(* CoDeSys 2.3 export: ALL.EXP *)
(* Libraries: ANALYZATION.LIB 5.10.99 08:05:06, G:\owen\dz_smarthome_lib.lib 9.5.15 16:30:44, G:\owen\lib\oscat_basic_333.lib 19.12.17 20:17:33, IECSFC.LIB 13.4.06 14:51:28, STANDARD.LIB 4.10.05 10:14:46, SysLibSockets.lib 20.2.06 13:31:14, SysLibTime.lib 20.2.06 13:31:16, Util.lib 18.5.10 14:14:28 *)

(* PLC configuration (modules and I/O channels)
PLC110_30 [Root] node -1, in %IB0 out %QB0 {param 1 = 1; param 2 = 1000; param 3 = 6}
  Fast discrete inputs [I_SIMPLE_INPUT] node 0, in %IB0 out %QB0 {param 1 = 10; param 9 = No}
    AT %IX0.0 [BitInput] Discrete input 1
    AT %IX0.1 [BitInput] Discrete input 2
  Discrete inputs - 16 [ID130] node 1, in %IB1 out %QB1 {param 1 = 1; param 9 = No; param 10 = 16}
    AT %IB1.0 [ByteInput] 8 discrete inputs
    AT %IB1.1 [ByteInput] 8 discrete inputs
  Fast discrete outputs [OWEN_ID570] node 2, in %IB2 out %QB2 {param 1 = FALSE; param 2 = FALSE; param 3 = FALSE; param 4 = FALSE; param 10 = No}
    RADIATOR_GUEST_OUT AT %QX2.0 [BitOutput] Fast discrete output 1 - radiator, guest room, 1 = OFF!
    RADIATOR_CHILDREN_NEAR_OUT AT %QX2.1 [BitOutput] Fast discrete output 2, radiator, children room, near the door, 1 = OFF
    RADIATOR_BEDROOM_OUT AT %QX2.2 [BitOutput] Fast discrete output 3
    RADIATOR_DINNER_OUT AT %QX2.3 [BitOutput] Fast discrete output 4 - dinner room radiator PWM, 0 = ON, 1 = OFF
  Discrete outputs - 8 [ID131] node 3, in %IB3 out %QB3 {param 1 = 0; param 4 = No; param 5 = 10}
    AT %QB3.0 [ByteOutput] 8 discrete outputs
  Special input [ID103] node 4, in %IB4 out %QB4 {param 1 = 1000; param 2 = 1; param 3 = 400; param 4 = 3000; param 5 = No}
    AT %IX4.0 [BitInput] Special input
  Special output [ID104] node 5, in %IB5 out %QB5 {param 1 = No; param 2 = 1}
    AT %QX5.0 [BitOutput] Special output
  ModBus (Master) [MODBUS_MASTER_ID450] node 6, in %IB6 out %QB6 {param 1 = No}
    AT %QD6.0 [DWordOutput] Last address
    AT %QW6.1 [WordOutput] Last error
    RS-485-1 [COM1_USART] node 0, in %IB6.0 out %QB6.0 {param 1 = 11520; param 2 = NO PARITY CHECK; param 3 = 8 bits; param 4 = One stop bit; param 5 = RS485; param 6 = ASCII; param 7 = 0; param 8 = No}
    OWEN_MVA8 [ID2050] node 1, in %IB6.1 out %QB6.1 {param 1 = 10:0:0:223; param 2 = 30; param 3 = 502; param 4 = Serial; param 5 = 80; param 6 = By poll time; param 7 = 400; param 8 = No; param 9 = 0; param 10 = Trace_mode}
      mva8_0_cmd AT %QB6.1.0 [ComChannel] Command (0xff - Start)
      Cycle time measuring on input 1 [ID2066] node 0, in %IB6.1.0 out %QB6.1.0 {param 1 = 3; param 2 = Command Read (03); param 7 = No}
        AT %IW6.1.0.0 [WordInput]
      Value in input 1 [ID2067] node 1, in %IB6.1.1 out %QB6.1.1 {param 1 = 4; param 2 = Command Read (03); param 7 = No}
        mva0_t0 AT %ID6.1.1.0 [FloatInput]
      Cycle time measuring on input 2 [ID2068] node 2, in %IB6.1.2 out %QB6.1.2 {param 1 = 9; param 2 = Command Read (03); param 7 = No}
        AT %IW6.1.2.0 [WordInput]
      Value in input 2 [ID2069] node 3, in %IB6.1.3 out %QB6.1.3 {param 1 = 10; param 2 = Command Read (03); param 7 = No}
        mva0_t1 AT %ID6.1.3.0 [FloatInput]
      Cycle time measuring on input 3 [ID2070] node 4, in %IB6.1.4 out %QB6.1.4 {param 1 = 15; param 2 = Command Read (03); param 7 = No}
        AT %IW6.1.4.0 [WordInput]
      Value in input 3 [ID2071] node 5, in %IB6.1.5 out %QB6.1.5 {param 1 = 16; param 2 = Command Read (03); param 7 = No}
        mva0_t2 AT %ID6.1.5.0 [FloatInput]
      Cycle time measuring on input 4 [ID2072] node 6, in %IB6.1.6 out %QB6.1.6 {param 1 = 21; param 2 = Command Read (03); param 7 = No}
        AT %IW6.1.6.0 [WordInput]
      Value in input 4 [ID2073] node 7, in %IB6.1.7 out %QB6.1.7 {param 1 = 22; param 2 = Command Read (03); param 7 = No}
        mva0_t3 AT %ID6.1.7.0 [FloatInput]
      Cycle time measuring on input 5 [ID2074] node 8, in %IB6.1.8 out %QB6.1.8 {param 1 = 27; param 2 = Command Read (03); param 7 = No}
        AT %IW6.1.8.0 [WordInput]
      Value in input 5 [ID2075] node 9, in %IB6.1.9 out %QB6.1.9 {param 1 = 28; param 2 = Command Read (03); param 7 = No}
        mva0_t4 AT %ID6.1.9.0 [FloatInput]
      Cycle time measuring on input 6 [ID2076] node 10, in %IB6.1.10 out %QB6.1.10 {param 1 = 33; param 2 = Command Read (03); param 7 = No}
        AT %IW6.1.10.0 [WordInput]
      Value in input 6 [ID2077] node 11, in %IB6.1.11 out %QB6.1.11 {param 1 = 34; param 2 = Command Read (03); param 7 = No}
        mva0_t5 AT %ID6.1.11.0 [FloatInput]
      Cycle time measuring on input 7 [ID2078] node 12, in %IB6.1.12 out %QB6.1.12 {param 1 = 39; param 2 = Command Read (03); param 7 = No}
        AT %IW6.1.12.0 [WordInput]
      Value in input 7 [ID2079] node 13, in %IB6.1.13 out %QB6.1.13 {param 1 = 40; param 2 = Command Read (03); param 7 = No}
        mva0_t6 AT %ID6.1.13.0 [FloatInput]
      Cycle time measuring on input 8 [ID2080] node 14, in %IB6.1.14 out %QB6.1.14 {param 1 = 45; param 2 = Command Read (03); param 7 = No}
        AT %IW6.1.14.0 [WordInput]
      Value in input 8 [ID2081] node 15, in %IB6.1.15 out %QB6.1.15 {param 1 = 46; param 2 = Command Read (03); param 7 = No}
        mva0_t7 AT %ID6.1.15.0 [FloatInput]
    OWEN_MVA8 [ID2050] node 2, in %IB6.2 out %QB6.2 {param 1 = 10:0:0:223; param 2 = 30; param 3 = 502; param 4 = Serial; param 5 = 88; param 6 = By poll time; param 7 = 400; param 8 = No; param 9 = 0; param 10 = Trace_mode}
      mva8_1_cmd AT %QB6.2.0 [ComChannel] Command (0xff - Start)
      Cycle time measuring on input 1 [ID2066] node 0, in %IB6.2.0 out %QB6.2.0 {param 1 = 3; param 2 = Command Read (03); param 7 = No}
        AT %IW6.2.0.0 [WordInput]
      Value in input 1 [ID2067] node 1, in %IB6.2.1 out %QB6.2.1 {param 1 = 4; param 2 = Command Read (03); param 7 = No}
        mva1_t0 AT %ID6.2.1.0 [FloatInput]
      Cycle time measuring on input 2 [ID2068] node 2, in %IB6.2.2 out %QB6.2.2 {param 1 = 9; param 2 = Command Read (03); param 7 = No}
        AT %IW6.2.2.0 [WordInput]
      Value in input 2 [ID2069] node 3, in %IB6.2.3 out %QB6.2.3 {param 1 = 10; param 2 = Command Read (03); param 7 = No}
        mva1_t1 AT %ID6.2.3.0 [FloatInput]
      Cycle time measuring on input 3 [ID2070] node 4, in %IB6.2.4 out %QB6.2.4 {param 1 = 15; param 2 = Command Read (03); param 7 = No}
        AT %IW6.2.4.0 [WordInput]
      Value in input 3 [ID2071] node 5, in %IB6.2.5 out %QB6.2.5 {param 1 = 16; param 2 = Command Read (03); param 7 = No}
        mva1_t2 AT %ID6.2.5.0 [FloatInput]
      Cycle time measuring on input 4 [ID2072] node 6, in %IB6.2.6 out %QB6.2.6 {param 1 = 21; param 2 = Command Read (03); param 7 = No}
        AT %IW6.2.6.0 [WordInput]
      Value in input 4 [ID2073] node 7, in %IB6.2.7 out %QB6.2.7 {param 1 = 22; param 2 = Command Read (03); param 7 = No}
        mva1_t3 AT %ID6.2.7.0 [FloatInput]
      Cycle time measuring on input 5 [ID2074] node 8, in %IB6.2.8 out %QB6.2.8 {param 1 = 27; param 2 = Command Read (03); param 7 = No}
        AT %IW6.2.8.0 [WordInput]
      Value in input 5 [ID2075] node 9, in %IB6.2.9 out %QB6.2.9 {param 1 = 28; param 2 = Command Read (03); param 7 = No}
        mva1_t4 AT %ID6.2.9.0 [FloatInput]
      Cycle time measuring on input 6 [ID2076] node 10, in %IB6.2.10 out %QB6.2.10 {param 1 = 33; param 2 = Command Read (03); param 7 = No}
        AT %IW6.2.10.0 [WordInput]
      Value in input 6 [ID2077] node 11, in %IB6.2.11 out %QB6.2.11 {param 1 = 34; param 2 = Command Read (03); param 7 = No}
        mva1_t5 AT %ID6.2.11.0 [FloatInput]
      Cycle time measuring on input 7 [ID2078] node 12, in %IB6.2.12 out %QB6.2.12 {param 1 = 39; param 2 = Command Read (03); param 7 = No}
        AT %IW6.2.12.0 [WordInput]
      Value in input 7 [ID2079] node 13, in %IB6.2.13 out %QB6.2.13 {param 1 = 40; param 2 = Command Read (03); param 7 = No}
        mva1_t6 AT %ID6.2.13.0 [FloatInput]
      Cycle time measuring on input 8 [ID2080] node 14, in %IB6.2.14 out %QB6.2.14 {param 1 = 45; param 2 = Command Read (03); param 7 = No}
        AT %IW6.2.14.0 [WordInput]
      Value in input 8 [ID2081] node 15, in %IB6.2.15 out %QB6.2.15 {param 1 = 46; param 2 = Command Read (03); param 7 = No}
        mva1_t7 AT %ID6.2.15.0 [FloatInput]
    OWEN_MVA8 [ID2050] node 3, in %IB6.3 out %QB6.3 {param 1 = 10:0:0:223; param 2 = 30; param 3 = 502; param 4 = Serial; param 5 = 96; param 6 = By poll time; param 7 = 400; param 8 = No; param 9 = 0; param 10 = Trace_mode}
      mva8_2_cmd AT %QB6.3.0 [ComChannel] Command (0xff - Start)
      Cycle time measuring on input 1 [ID2066] node 0, in %IB6.3.0 out %QB6.3.0 {param 1 = 3; param 2 = Command Read (03); param 7 = No}
        AT %IW6.3.0.0 [WordInput]
      Value in input 1 [ID2067] node 1, in %IB6.3.1 out %QB6.3.1 {param 1 = 4; param 2 = Command Read (03); param 7 = No}
        mva2_t0 AT %ID6.3.1.0 [FloatInput]
      Cycle time measuring on input 2 [ID2068] node 2, in %IB6.3.2 out %QB6.3.2 {param 1 = 9; param 2 = Command Read (03); param 7 = No}
        AT %IW6.3.2.0 [WordInput]
      Value in input 2 [ID2069] node 3, in %IB6.3.3 out %QB6.3.3 {param 1 = 10; param 2 = Command Read (03); param 7 = No}
        mva2_t1 AT %ID6.3.3.0 [FloatInput]
      Cycle time measuring on input 3 [ID2070] node 4, in %IB6.3.4 out %QB6.3.4 {param 1 = 15; param 2 = Command Read (03); param 7 = No}
        AT %IW6.3.4.0 [WordInput]
      Value in input 3 [ID2071] node 5, in %IB6.3.5 out %QB6.3.5 {param 1 = 16; param 2 = Command Read (03); param 7 = No}
        mva2_t2 AT %ID6.3.5.0 [FloatInput]
      Cycle time measuring on input 4 [ID2072] node 6, in %IB6.3.6 out %QB6.3.6 {param 1 = 21; param 2 = Command Read (03); param 7 = No}
        AT %IW6.3.6.0 [WordInput]
      Value in input 4 [ID2073] node 7, in %IB6.3.7 out %QB6.3.7 {param 1 = 22; param 2 = Command Read (03); param 7 = No}
        mva2_t3 AT %ID6.3.7.0 [FloatInput]
      Cycle time measuring on input 5 [ID2074] node 8, in %IB6.3.8 out %QB6.3.8 {param 1 = 27; param 2 = Command Read (03); param 7 = No}
        AT %IW6.3.8.0 [WordInput]
      Value in input 5 [ID2075] node 9, in %IB6.3.9 out %QB6.3.9 {param 1 = 28; param 2 = Command Read (03); param 7 = No}
        mva2_t4 AT %ID6.3.9.0 [FloatInput]
      Cycle time measuring on input 6 [ID2076] node 10, in %IB6.3.10 out %QB6.3.10 {param 1 = 33; param 2 = Command Read (03); param 7 = No}
        AT %IW6.3.10.0 [WordInput]
      Value in input 6 [ID2077] node 11, in %IB6.3.11 out %QB6.3.11 {param 1 = 34; param 2 = Command Read (03); param 7 = No}
        mva2_t5 AT %ID6.3.11.0 [FloatInput]
      Cycle time measuring on input 7 [ID2078] node 12, in %IB6.3.12 out %QB6.3.12 {param 1 = 39; param 2 = Command Read (03); param 7 = No}
        AT %IW6.3.12.0 [WordInput]
      Value in input 7 [ID2079] node 13, in %IB6.3.13 out %QB6.3.13 {param 1 = 40; param 2 = Command Read (03); param 7 = No}
        mva2_t6 AT %ID6.3.13.0 [FloatInput]
      Cycle time measuring on input 8 [ID2080] node 14, in %IB6.3.14 out %QB6.3.14 {param 1 = 45; param 2 = Command Read (03); param 7 = No}
        AT %IW6.3.14.0 [WordInput]
      Value in input 8 [ID2081] node 15, in %IB6.3.15 out %QB6.3.15 {param 1 = 46; param 2 = Command Read (03); param 7 = No}
        mva2_t7 AT %ID6.3.15.0 [FloatInput]
  ModBus (Master) [MODBUS_MASTER_ID450] node 7, in %IB7 out %QB7 {param 1 = No}
    AT %QD7.0 [DWordOutput] Last address
    AT %QW7.1 [WordOutput] Last error
    RS-485-2 [COM3_USART] node 0, in %IB7.0 out %QB7.0 {param 1 = 9600; param 2 = NO PARITY CHECK; param 3 = 8 bits; param 4 = One stop bit; param 5 = RS485; param 6 = RTU; param 7 = 0; param 8 = No}
    Universal Modbus device [ID2000] node 1, in %IB7.1 out %QB7.1 {param 1 = 10:0:0:223; param 2 = 150; param 3 = 502; param 4 = Serial; param 5 = 16; param 6 = By value change; param 7 = 200; param 8 = No; param 9 = 0; param 10 = Trace_mode}
      z033_special_cmd AT %QB7.1.0 [ComChannel] Command (0xff - Start)
      Register output module [ID2004] node 0, in %IB7.1.0 out %QB7.1.0 {param 1 = 16#116; param 2 = Preset singl register (0x06); param 8 = No}
        z033_hum116_out AT %QW7.1.0.0 [WordOutput]
      Register output module [ID2004] node 1, in %IB7.1.1 out %QB7.1.1 {param 1 = 16#115; param 2 = Preset singl register (0x06); param 8 = No}
        z033_temperature115_out AT %QW7.1.1.0 [WordOutput]
    Universal Modbus device [ID2000] node 2, in %IB7.2 out %QB7.2 {param 1 = 10:0:0:223; param 2 = 150; param 3 = 502; param 4 = Serial; param 5 = 16; param 6 = Both; param 7 = 200; param 8 = No; param 9 = 0; param 10 = Trace_mode}
      z033_cmd AT %QB7.2.0 [ComChannel] Command (0xff - Start)
      Register output module [ID2004] node 0, in %IB7.2.0 out %QB7.2.0 {param 1 = 16#112; param 2 = Preset singl register (0x06); param 8 = No}
        z033_Setup112 AT %QW7.2.0.0 [WordOutput]
      Register output module [ID2004] node 1, in %IB7.2.1 out %QB7.2.1 {param 1 = 16#113; param 2 = Preset singl register (0x06); param 8 = No}
        z033_Setup113 AT %QW7.2.1.0 [WordOutput]
      Register input module [ID2003] node 2, in %IB7.2.2 out %QB7.2.2 {param 1 = 16#114; param 2 = Read holding Registers  (0x03); param 8 = No}
        z033_mode114_in AT %IW7.2.2.0 [WordInput]
      Register output module [ID2004] node 3, in %IB7.2.3 out %QB7.2.3 {param 1 = 16#114; param 2 = Preset singl register (0x06); param 8 = No}
        z033_mode114_out AT %QW7.2.3.0 [WordOutput]
      Register input module [ID2003] node 4, in %IB7.2.4 out %QB7.2.4 {param 1 = 16#115; param 2 = Read holding Registers  (0x03); param 8 = No}
        z033_temperature115_in AT %IW7.2.4.0 [WordInput]
      Register input module [ID2003] node 5, in %IB7.2.5 out %QB7.2.5 {param 1 = 16#116; param 2 = Read holding Registers  (0x03); param 8 = No}
        z033_hum116_in AT %IW7.2.5.0 [WordInput]
      Register input module [ID2003] node 6, in %IB7.2.6 out %QB7.2.6 {param 1 = 16#117; param 2 = Read holding Registers  (0x03); param 8 = No}
        z033_room_temp117_in AT %IW7.2.6.0 [WordInput] temp measured by panel, no set
      Register output module [ID2004] node 7, in %IB7.2.7 out %QB7.2.7 {param 1 = 16#118; param 2 = Preset singl register (0x06); param 8 = No}
        z033_floor_temp118_out AT %QW7.2.7.0 [WordOutput]
      Register output module [ID2004] node 8, in %IB7.2.8 out %QB7.2.8 {param 1 = 16#119; param 2 = Preset singl register (0x06); param 8 = No}
        z033_outdoor_hum119_out AT %QW7.2.8.0 [WordOutput]
      Register output module [ID2004] node 9, in %IB7.2.9 out %QB7.2.9 {param 1 = 16#11A; param 2 = Preset singl register (0x06); param 8 = No}
        z033_room_hum11a_out AT %QW7.2.9.0 [WordOutput]
      Register output module [ID2004] node 10, in %IB7.2.10 out %QB7.2.10 {param 1 = 16#11B; param 2 = Preset singl register (0x06); param 8 = No}
        z033_air_hum11b_out AT %QW7.2.10.0 [WordOutput]
      Register output module [ID2004] node 11, in %IB7.2.11 out %QB7.2.11 {param 1 = 16#11c; param 2 = Preset singl register (0x06); param 8 = No}
        z033_errmode11c_out AT %QW7.2.11.0 [WordOutput]
      Register output module [ID2004] node 12, in %IB7.2.12 out %QB7.2.12 {param 1 = 16#11D; param 2 = Preset singl register (0x06); param 8 = No}
        z033_clock11d_out AT %QW7.2.12.0 [WordOutput]
      Register input module [ID2003] node 13, in %IB7.2.13 out %QB7.2.13 {param 1 = 16#11C; param 2 = Read holding Registers  (0x03); param 8 = No}
        z033_errmode11c_in AT %IW7.2.13.0 [WordInput]
      Register output module [ID2004] node 14, in %IB7.2.14 out %QB7.2.14 {param 1 = 16#117; param 2 = Preset singl register (0x06); param 8 = No}
        z033_air_temp_117_out AT %QW7.2.14.0 [WordOutput]
  Button [ID003] node 8, in %IB8 out %QB8
    AT %IX8.0 [BitInput] Button Start/Stop
  ModBus (slave) [MODBUS_ID400] node 9, in %IB9 out %QB9 {param 1 = 1; param 2 = No}
    Modbus [MODBUS_ID302] node 0, in %IB9.0 out %QB9.0
      TCP [TCP_ID221] node 0, in %IB9.0.0 out %QB9.0.0 {param 1 = 502; param 2 = No}
    2 byte [Register] node 1, in %IB9.1 out %QB9.1
      Uplink_Target_Temp AT %QW9.1.0 [WordOutput]
    2 byte [Register] node 2, in %IB9.2 out %QB9.2
      Uplink_Target_Humid AT %QW9.2.0 [WordOutput]
  ModBus (Master) [MODBUS_MASTER_ID450] node 10, in %IB10 out %QB10 {param 1 = No}
    AT %QD10.0 [DWordOutput] Last address
    AT %QW10.1 [WordOutput] Last error
    Debug RS-232 [DEBUG_USART] node 0, in %IB10.0 out %QB10.0 {param 1 = 11520; param 2 = NO PARITY CHECK; param 3 = 8 bits; param 4 = One stop bit; param 5 = RS232; param 6 = ASCII; param 7 = 0; param 8 = No}
    Universal Modbus device [ID2000] node 1, in %IB10.1 out %QB10.1 {param 1 = 192:168:88:130; param 2 = 150; param 3 = 502; param 4 = TCP; param 5 = 1; param 6 = By poll time; param 7 = 2000; param 8 = No; param 9 = 0; param 10 = Trace_mode}
      dz1w_cmd AT %QB10.1.0 [ComChannel] Command (0xff - Start)
      Register input module [ID2003] node 0, in %IB10.1.0 out %QB10.1.0 {param 1 = 1024; param 2 = Read holding Registers  (0x03); param 8 = No}
        sensor_id0 AT %IW10.1.0.0 [WordInput]
      Register input module [ID2003] node 1, in %IB10.1.1 out %QB10.1.1 {param 1 = 1025; param 2 = Read holding Registers  (0x03); param 8 = No}
        sensor_id1 AT %IW10.1.1.0 [WordInput]
      Register input module [ID2003] node 2, in %IB10.1.2 out %QB10.1.2 {param 1 = 1026; param 2 = Read holding Registers  (0x03); param 8 = No}
        sensor_id2 AT %IW10.1.2.0 [WordInput]
      Register input module [ID2003] node 3, in %IB10.1.3 out %QB10.1.3 {param 1 = 1027; param 2 = Read holding Registers  (0x03); param 8 = No}
        sensor_id3 AT %IW10.1.3.0 [WordInput]
      Register input module [ID2003] node 4, in %IB10.1.4 out %QB10.1.4 {param 1 = 1028; param 2 = Read holding Registers  (0x03); param 8 = No}
        sensor_id4 AT %IW10.1.4.0 [WordInput]
      Register input module [ID2003] node 5, in %IB10.1.5 out %QB10.1.5 {param 1 = 1029; param 2 = Read holding Registers  (0x03); param 8 = No}
        sensor_id5 AT %IW10.1.5.0 [WordInput]
      Register input module [ID2003] node 6, in %IB10.1.6 out %QB10.1.6 {param 1 = 1030; param 2 = Read holding Registers  (0x03); param 8 = No}
        sensor_id6 AT %IW10.1.6.0 [WordInput]
      Register input module [ID2003] node 7, in %IB10.1.7 out %QB10.1.7 {param 1 = 1031; param 2 = Read holding Registers  (0x03); param 8 = No}
        sensor_id7 AT %IW10.1.7.0 [WordInput]
      Register input module [ID2003] node 8, in %IB10.1.8 out %QB10.1.8 {param 1 = 1032; param 2 = Read holding Registers  (0x03); param 8 = No}
        sensor_id8 AT %IW10.1.8.0 [WordInput]
      Register input module [ID2003] node 9, in %IB10.1.9 out %QB10.1.9 {param 1 = 1033; param 2 = Read holding Registers  (0x03); param 8 = No}
        sensor_id9 AT %IW10.1.9.0 [WordInput]
      Register input module [ID2003] node 10, in %IB10.1.10 out %QB10.1.10 {param 1 = 1034; param 2 = Read holding Registers  (0x03); param 8 = No}
        sensor_id10 AT %IW10.1.10.0 [WordInput]
      Register input module [ID2003] node 11, in %IB10.1.11 out %QB10.1.11 {param 1 = 2048; param 2 = Read holding Registers  (0x03); param 8 = No}
        seq_sensor_0 AT %IW10.1.11.0 [WordInput]
      Register input module [ID2003] node 12, in %IB10.1.12 out %QB10.1.12 {param 1 = 2049; param 2 = Read holding Registers  (0x03); param 8 = No}
        seq_sensor_1 AT %IW10.1.12.0 [WordInput]
*)

(* Task configuration *)
TASK OnceASecond (PRIORITY := 1, INTERVAL := T#1s0ms);
ONCE_A_SECOND_PRG();
END_TASK
TASK HTTP_POLLER (PRIORITY := 5, INTERVAL := T#1s0ms);
TCP_POLL();
END_TASK
TASK Main (PRIORITY := 2, INTERVAL := T#50ms);
PLC_PRG();
END_TASK
TASK MQTT (PRIORITY := 4, INTERVAL := T#1s0ms);
MQTT_MAIN();
END_TASK

(* Global variable list: Global_Variables *)
VAR_GLOBAL RETAIN PERSISTENT


	GLOBAL_Target_Room_Temp				: REAL := 26;
	GLOBAL_Target_Room_Humid				: REAL := 30;

	GLOBAL_Current_Entrance_Air_Temp		: REAL	:= 0;
	GLOBAL_Current_Entrance_Floor_Temp	: REAL := 100;

	GLOBAL_Current_Bath_Air_Temp			: REAL	:= 0;
	GLOBAL_Current_Bath_Floor_Temp		: REAL := 100;

	GLOBAL_Current_Bath_Tube_Temp		: REAL := 0;

	GLOBAL_Current_Dinner_Air_Temp			: REAL	:= 0;		(* Composite made of 3 sensors, used to control floor *)
	GLOBAL_Current_Dinner_Floor_Temp		: REAL := 100;

	GLOBAL_Current_Dinner_Air_Bottom_Temp			: REAL	:= 0; (* Bottom sensor, near the radiator *)
	GLOBAL_Current_Dinner_Air_Middle_Temp			: REAL	:= 0; (* Middle sensor, in the z033 panel, 1 degree step *)

	GLOBAL_Current_Guest_Air_Temp			: REAL := 0;

	GLOBAL_Current_Kitchen_Air_Ceiling_Temp			: REAL	:= 0; (* Ceiling sensor, in the fire sensor, kitchen *)

	GLOBAL_Current_Children_Air_Temp		: REAL	:= 0;
	GLOBAL_Current_Children_Floor_Temp	: REAL := 100;

	GLOBAL_Current_Badroom_Air_Temp		: REAL	:= 0;

	GLOBAL_Current_Bath_Air_Humid			: REAL := 0;

	GLOBAL_Current_Outdoor_Air_Temp		: REAL := 0;


END_VAR



VAR_GLOBAL CONSTANT
	SANE_TEMP_MIN: REAL := 10;		(*Minimum temp value assumed to be sane*)
	SANE_TEMP_MAX: REAL := 40;		(*Maximum temp value assumed to be sane*)

	SANE_HUMID_MIN:	WORD		:= 15;
	SANE_HUMID_MAX:	WORD		:= 55;

END_VAR

(* POU ONCE_A_SECOND_PRG, ST *)
PROGRAM ONCE_A_SECOND_PRG

VAR

	FLOOR_ENTRANCE		: FLOOR_PID;
	FLOOR_BATH				: FLOOR_PID;
	(*FLOOR_DINNER			: FLOOR_PID;*)
	DINNER_PID			: DUAL_PID;
	(*FLOOR_CHILDREN		: FLOOR_PID;*)
	CHILDREN_PID			: DUAL_PID;
	GUEST_PID			: DUAL_PID;

	PWM_ENTRANCE		: PWM;
	PWM_BATH				: PWM;
	PWM_DINNER			: PWM;
	PWM_CHILDREN			: PWM;

(*	PWM_DINNER_RADIATOR		: PWM; *)
	PWM_DINNER_RADIATOR		: RADIATOR_PWM;
	PWM_GUEST_RADIATOR		: RADIATOR_PWM;
	PWM_CHILDREN_RADIATOR	: RADIATOR_PWM;


END_VAR
	(* Must be called once a second! *)



	(* Entrance *)

	FLOOR_ENTRANCE( Target := GLOBAL_Target_Room_Temp, Current := GLOBAL_Current_Entrance_Air_Temp, Floor := GLOBAL_Current_Entrance_Floor_Temp );

	PWM_ENTRANCE( DUTY := FLOOR_ENTRANCE.DUTY, PHASE_SHIFT := 0 );

	HEAT_ENTRANCE_OUT := PWM_ENTRANCE.OUT_ON;



	(* Bath *)

	FLOOR_BATH( Target := GLOBAL_Target_Room_Temp, Current := GLOBAL_Current_Bath_Air_Temp, Floor := GLOBAL_Current_Bath_Floor_Temp );

	PWM_BATH( DUTY := FLOOR_BATH.DUTY, PHASE_SHIFT := 2 );

	HEAT_BATH_OUT := PWM_BATH.OUT_ON;


	(* Dinner *)

(*
	FLOOR_DINNER( Target := GLOBAL_Target_Room_Temp, Current := GLOBAL_Current_Dinner_Air_Temp, Floor := GLOBAL_Current_Dinner_Floor_Temp );
*)
	DINNER_PID( Target := GLOBAL_Target_Room_Temp, Current := GLOBAL_Current_Dinner_Air_Temp, Floor := GLOBAL_Current_Dinner_Floor_Temp );

	PWM_DINNER( DUTY := DINNER_PID.FLOOR_DUTY, PHASE_SHIFT := 4 );

	PWM_DINNER_RADIATOR( DUTY := DINNER_PID.RADIATOR_DUTY, PHASE_SHIFT := 0 );

	HEAT_DINNER_OUT := PWM_DINNER.OUT_ON;

	RADIATOR_DINNER_OUT := NOT PWM_DINNER_RADIATOR.OUT_ON; (* Naive impl - just control radiator just like floor *)

	(* Guest - no hot floor *)

	GUEST_PID( Target := GLOBAL_Target_Room_Temp, Current := GLOBAL_Current_Guest_Air_Temp, Floor := 50 ); (* no floor, give insane input value *)
	PWM_GUEST_RADIATOR( DUTY := GUEST_PID.RADIATOR_DUTY, PHASE_SHIFT := 0 );
	RADIATOR_GUEST_OUT := NOT PWM_GUEST_RADIATOR.OUT_ON; (* Naive impl - just control radiator just like floor *)

	(* Children *)

	(* FLOOR_CHILDREN( Target := GLOBAL_Target_Room_Temp, Current := GLOBAL_Current_CHILDREN_Air_Temp, Floor := GLOBAL_Current_CHILDREN_Floor_Temp ); *)

	CHILDREN_PID(        Target := GLOBAL_Target_Room_Temp, Current := GLOBAL_Current_CHILDREN_Air_Temp, Floor := GLOBAL_Current_CHILDREN_Floor_Temp );

	(*PWM_CHILDREN( DUTY := FLOOR_CHILDREN.DUTY, PHASE_SHIFT := 6 );*)
	PWM_CHILDREN( DUTY := CHILDREN_PID.FLOOR_DUTY, PHASE_SHIFT := 6 );


	PWM_CHILDREN_RADIATOR( DUTY := CHILDREN_PID.RADIATOR_DUTY, PHASE_SHIFT := 0 );

	HEAT_CHILDREN_OUT := PWM_CHILDREN.OUT_ON;

	RADIATOR_CHILDREN_NEAR_OUT := NOT PWM_CHILDREN_RADIATOR.OUT_ON;
END_PROGRAM

(* POU PID-PWM/FLOOR_PID, ST *)
FUNCTION_BLOCK FLOOR_PID

VAR_INPUT
	Target			: REAL;		(* Уставка, target ROOM temperature value to achieve *)
	Current		: REAL;		(* Current measured ROOM temperature value *)

	Floor			: REAL;		(* Current measured FLOOR temperature value *)
	Limited		: REAL := 35;	(* maximum FLOOR temperature value not to overcome*)


END_VAR

VAR_OUTPUT

	DUTY				: INT;		(* Duty cycle for heater *)

END_VAR

VAR

	TMP				: INT;
(*
	INTEGRAL			: INT;
*)
END_VAR
(*

	Actually we have TWO regulators here, one is PID (or PI) - for room temperature,
	and one is simple limiting for floor temperature.

*)

	(* room temp seems to be insane, use floor temp instead *)
	IF Current < 1 THEN
		Current := Floor;
	END_IF


	(* Simple FLOOR temp limit *)

	IF Floor > Limited THEN
		DUTY := 0;
		RETURN;
	END_IF

	(* TEMPORARY IMPL! *)

	IF Current > Target THEN
		DUTY := 0;
		RETURN;
	END_IF

	TMP := REAL_TO_INT(  (Target - Current) * 100 / 4 ); (* 4 degrees of difference mean 100% of power *)

	IF TMP < 0 THEN
		TMP := 0;
	END_IF

	IF TMP > 100 THEN
		TMP := 100;
	END_IF

	DUTY := TMP;
END_FUNCTION_BLOCK

(* POU PID-PWM/DUAL_PID, ST *)
FUNCTION_BLOCK DUAL_PID

VAR_INPUT
	Target			: REAL;		(* Уставка, target ROOM temperature value to achieve *)
	Current		: REAL;		(* Current measured ROOM temperature value *)

	Floor			: REAL;		(* Current measured FLOOR temperature value *)
	Limited		: REAL := 33;	(* Maximum FLOOR temperature value not to overcome*)


END_VAR

VAR_OUTPUT

	FLOOR_DUTY				: INT;		(* Duty cycle for floor heater *)
	RADIATOR_DUTY				: INT;		(* Duty cycle for wall radiator *)

END_VAR

VAR

	LINEAR			: INT;
	INTEGRAL			: REAL;		(* +- 1000 *)
	DIFFERENTIAL 	: REAL;		(* +- 100 *)
	DUTY				: INT;		(* Duty cycle - total *)

	Diff_Timer			: INT;
	Diff_Prev_Temp	: REAL		:= -1000;
	Diff_Temp_Delta	: REAL;		(* Difference of temperature in one minute *)
	Diff_Sane 			: BOOL;

END_VAR


VAR CONSTANT

	ONLY_RADIATOR_DUTY_LIMIT	: INT := 20;

	Diff_Timer_Time					: INT := 120;

END_VAR
(*

	Actually we have TWO regulators here, one is PID (or PI) - for room temperature,
	and one is simple limiting for floor temperature.

*)

	(* room temp seems to be insane, use floor temp instead *)
	IF Current < 1 THEN
		Current := Floor;
	END_IF




	LINEAR := REAL_TO_INT(  (Target - Current) * 100 / 4 ); (* 4 degrees of difference mean 100% of power *)
	LINEAR := REAL_TO_INT( LIMIT_VALUE( LINEAR, -100, 100) );

	(* Integral part *)

	INTEGRAL := INTEGRAL + (LINEAR / 2500.0); (* integration time about 0,65 hr *)

	INTEGRAL := LIMIT_VALUE( INTEGRAL, -100, 100 );

	(* Diff part *)

	Diff_Sane := TRUE;

	Diff_Timer := Diff_Timer + 1;
	IF Diff_Timer >= Diff_Timer_Time THEN
		Diff_Timer := 0;

		IF NOT IS_SANE_TEMP( Diff_Prev_Temp ) THEN
			Diff_Sane := FALSE;
		END_IF

		Diff_Temp_Delta := Current - Diff_Prev_Temp;
		Diff_Prev_Temp := Current;

	END_IF

	IF NOT Diff_Sane THEN
		Diff_Temp_Delta := 0;
	END_IF

	(* MINUS 0.5 degree per 2 minutes is 400% of power *)
	DIFFERENTIAL := - Diff_Temp_Delta * 200 * 4;

	(* Limit diff part to 60% *)
	DIFFERENTIAL := LIMIT_VALUE( DIFFERENTIAL, 0, 60 );

	(* Common total integral + linear *)

	DUTY := LINEAR +  REAL_TO_INT (INTEGRAL/2); (* max integral part is 50% *)

	(* Just up - we're heating only *)

	DUTY := INT_LIMIT_VALUE( DUTY, 0, 100 );


	(* Radiator has 100% of integral part so that when we have major warmth loss we compensate it mostly with radiator *)
	RADIATOR_DUTY := DUTY + REAL_TO_INT (INTEGRAL/2);


	IF DUTY < ONLY_RADIATOR_DUTY_LIMIT THEN
		FLOOR_DUTY := 0;
	ELSE
		FLOOR_DUTY := (( DUTY- ONLY_RADIATOR_DUTY_LIMIT) * 100) / (100 - ONLY_RADIATOR_DUTY_LIMIT);
	END_IF


(*
	FLOOR_DUTY := DUTY;
	RADIATOR_DUTY := DUTY;
*)

	(* Add differential part just to floor power *)
	FLOOR_DUTY := FLOOR_DUTY + REAL_TO_INT(  DIFFERENTIAL );


	FLOOR_DUTY := INT_LIMIT_VALUE( FLOOR_DUTY, 0, 100 );
	RADIATOR_DUTY := INT_LIMIT_VALUE( RADIATOR_DUTY, 0, 100 );


	(* Simple FLOOR temp limit *)

	IF Floor > Limited THEN
		FLOOR_DUTY := 0;
	END_IF
END_FUNCTION_BLOCK

(* POU Conv/LIMIT_VALUE, ST *)
FUNCTION LIMIT_VALUE : REAL
VAR_INPUT
	V : REAL;
	MIN_V: REAL;
	MAX_V: REAL;
END_VAR

VAR
END_VAR
IF V > MAX_V THEN
	V := MAX_V;
END_IF

IF V < MIN_V THEN
	V := MIN_V;
END_IF

LIMIT_VALUE := V;
END_FUNCTION

(* POU Conv/IS_SANE_TEMP, ST *)
FUNCTION IS_SANE_TEMP : BOOL

VAR_INPUT
	T : REAL;
END_VAR

VAR
END_VAR
IF (T < SANE_TEMP_MIN) OR (T > SANE_TEMP_MAX) THEN
	IS_SANE_TEMP := FALSE;
ELSE
	IS_SANE_TEMP := TRUE;
END_IF
END_FUNCTION

(* POU Conv/INT_LIMIT_VALUE, ST *)
FUNCTION INT_LIMIT_VALUE : INT
VAR_INPUT
	V : INT;
	MIN_V: INT;
	MAX_V: INT;
END_VAR

VAR
END_VAR
IF V > MAX_V THEN
	V := MAX_V;
END_IF

IF V < MIN_V THEN
	V := MIN_V;
END_IF

INT_LIMIT_VALUE := V;
END_FUNCTION

(* POU PID-PWM/PWM, ST *)
FUNCTION_BLOCK PWM

VAR_INPUT
	DUTY 			: UINT;				(* 0-99, percent *)
	HI_VOLTAGE	: BOOL := FALSE; (* By default assume the heater is connected all the time *)
(*
	CYCLE_TIME	: TIME := t#10s;
*)

	PHASE_SHIFT	:	INT := 0;

END_VAR

VAR_OUTPUT
	OUT_ON				: BOOL := FALSE;
	LOAD_DETECTED	: BOOL := FALSE;
END_VAR

VAR
	On_Count				: INT := 0;

	Call_Count 			: INT := 0;
	Check_Load_Count	: INT := 0;	(* Once a while we do check for load to be connected *)

	Blinker					: BLINK;
	Blink_Once			: BOOL := FALSE;
END_VAR

VAR CONSTANT
	Check_Load_Count_Limit	: INT := 128;
	Cycle_Steps					: INT := 10;
END_VAR
(*

We assume that load (actual heater) can be disconnected with a wall switch.
We detect such a situation by turning power off and measuring voltage on heater.
(There must be a resistor over a relay contacts to provide some voltage)

HI_VOLTAGE is just for that.

*)

	(* Once a second *)

(* Called once a second anyway
	Blinker( TimeLow := t#0.5s, TimeHigh := t#0.5s, Enable := TRUE );

	IF NOT Blinker.OUT THEN
		Blink_Once := FALSE;
		RETURN;
	END_IF

	IF Blink_Once THEN
		RETURN;
	END_IF

	Blink_Once := TRUE;
*)
	(* Ok, next second came, do some task *)

	Call_Count := Call_Count + 1;  (* Count seconds *)

	IF NOT OUT_ON THEN (* Check for load *)
		Check_Load_Count := 0; (* No need to turn off - already off *)
		LOAD_DETECTED := NOT HI_VOLTAGE;
	END_IF

	Check_Load_Count := Check_Load_Count + 1;

	IF Check_Load_Count > Check_Load_Count_Limit THEN
		Check_Load_Count := 0;
		(* Override output to be off so that we will check if load is connected on next iteration *)
		OUT_ON := FALSE;
		RETURN;
	END_IF


	IF Call_Count > (Cycle_Steps-1 + PHASE_SHIFT) THEN
		Call_Count := 0 + PHASE_SHIFT;
		On_Count := (DUTY * Cycle_Steps) / 100;
	END_IF

	IF On_Count > 0 THEN
		OUT_ON := TRUE;
		On_Count := On_Count - 1;
	ELSE
		OUT_ON := FALSE;
	END_IF
END_FUNCTION_BLOCK

(* POU PID-PWM/RADIATOR_PWM, ST *)
FUNCTION_BLOCK RADIATOR_PWM

(**
 *		Thermal radiator actuator PWM drive.	Works with 24v SR actuator, normally open.
 *
 *		It seems that actuator really works within 0-20% of duty cycle, which means 80-100% for us.
**)


VAR_INPUT
	DUTY 				:	UINT;				(* 0-99, percent *)
	PHASE_SHIFT	:	INT		:= 0;
	ACTIVE			:	BOOL	:= TRUE;

END_VAR

VAR_OUTPUT
	OUT_ON				: BOOL := FALSE;
END_VAR

VAR
	On_Count				: INT := 0;
	Call_Count 			: INT := 0;

	Real_Duty				: INT := 0;

	Blinker					: BLINK;
	Blink_Once			: BOOL := FALSE;
END_VAR

VAR CONSTANT
	Cycle_Steps					: INT := 500; (* we need 500 sec cycle for radiator actuator *)
END_VAR
	(* Must be called once a second *)
	Call_Count := Call_Count + 1;  (* Count seconds *)

	(*Real_Duty := REAL_TO_INT( LIMIT_VALUE( (DUTY / 2) + 50, 0, 100 ) ); *)
	Real_Duty := REAL_TO_INT( DUTY );

	IF Call_Count > (Cycle_Steps-1 + PHASE_SHIFT) THEN
		Call_Count := 0 + PHASE_SHIFT;
		On_Count := (Real_Duty * Cycle_Steps) / 100;
	END_IF

	IF On_Count > 0 THEN
		OUT_ON := TRUE;
		On_Count := On_Count - 1;
	ELSE
		OUT_ON := FALSE;
	END_IF
END_FUNCTION_BLOCK

(* POU HTTP/TCP_POLL, ST *)
PROGRAM TCP_POLL

VAR

	HC		: HTTP_CLIENT;

END_VAR
IF TRUE THEN
	HC();
END_IF
END_PROGRAM

(* POU HTTP/HTTP_CLIENT, ST *)
FUNCTION_BLOCK HTTP_CLIENT
VAR_INPUT
END_VAR
VAR_OUTPUT
END_VAR

VAR

	m_dnSocket		:	DINT	:= SOCKET_INVALID;
(*	m_SAddress		:	SOCKADDRESS; *)

	m_error			:	INT		:= 0;

(*	o_dnRes			:	DINT; *)

	state				:	INT		:= 0;

	CONNECT		:	HTTP_CONNECT;

END_VAR

VAR CONSTANT
	wOutPort: INT := 8080;

	yOutAddr1: BYTE := 192;
	yOutAddr2: BYTE := 168;
	yOutAddr3: BYTE := 1;
	yOutAddr4: BYTE := 141;
(*	yOutAddr4: BYTE := 100; *)

(*
	yOutAddr4: BYTE := 192;
	yOutAddr3: BYTE := 168;
	yOutAddr2: BYTE := 1;
	yOutAddr1: BYTE := 100;
*)

	request: STRING := 'GET / HTTP/1.0$R$L$R$L';
END_VAR
	IF m_dnSocket = SOCKET_INVALID THEN

		CONNECT(  yOutAddr1:= yOutAddr1, yOutAddr2 := yOutAddr2, yOutAddr3 := yOutAddr3, yOutAddr4 := yOutAddr4, wOutPort := wOutPort, m_dnSocket := m_dnSocket, m_error := m_error  );
		RETURN; (* this shit needs some timeout between connect and send! *)

	END_IF


	CASE state  OF

	0:	HTTP_SEND_REAL( m_dnSocket, 'Current_Children_Floor_Temp', GLOBAL_Current_Children_Floor_Temp );
	1:	HTTP_SEND_REAL( m_dnSocket, 'Current_Children_Air_Temp', GLOBAL_Current_Children_Air_Temp );

	2:	HTTP_SEND_REAL( m_dnSocket, 'Current_Dinner_Floor_Temp', GLOBAL_Current_Dinner_Floor_Temp );
	3:	HTTP_SEND_REAL( m_dnSocket, 'Current_Dinner_Air_Temp', GLOBAL_Current_Dinner_Air_Temp );

	4:	HTTP_SEND_REAL( m_dnSocket, 'Current_Bath_Air_Temp', GLOBAL_Current_Bath_Air_Temp );
	5:	HTTP_SEND_REAL( m_dnSocket, 'Current_Bath_Floor_Temp', GLOBAL_Current_Bath_Floor_Temp );

	6:	HTTP_SEND_REAL( m_dnSocket, 'Current_Entrance_Air_Temp', GLOBAL_Current_Entrance_Air_Temp );
	7:	HTTP_SEND_REAL( m_dnSocket, 'Current_Entrance_Floor_Temp', GLOBAL_Current_Entrance_Floor_Temp );

	8:	HTTP_SEND_REAL( m_dnSocket, 'Current_Bath_Tube_Temp', GLOBAL_Current_Bath_Tube_Temp );

	9:	HTTP_SEND_REAL( m_dnSocket, 	'Current_Bath_Air_Humid', GLOBAL_Current_Bath_Air_Humid );

	10:	HTTP_SEND_REAL( m_dnSocket, 	'Current_Outdoor_Air_Temp', GLOBAL_Current_Outdoor_Air_Temp );

	11:	HTTP_SEND_REAL( m_dnSocket, 	'Current_Dinner_Air_Bottom_Temp', GLOBAL_Current_Dinner_Air_Bottom_Temp );
	12:	HTTP_SEND_REAL( m_dnSocket, 	'Current_Dinner_Air_Middle_Temp', GLOBAL_Current_Dinner_Air_Middle_Temp );

	13:	HTTP_SEND_REAL( m_dnSocket, 	'Current_Kitchen_Air_Ceiling_Temp', GLOBAL_Current_Kitchen_Air_Ceiling_Temp );

	14:	HTTP_SEND_REAL( m_dnSocket, 	'Current_Badroom_Air_Temp', GLOBAL_Current_Badroom_Air_Temp );

	ELSE
		state := -1;

		HTTP_SEND_REAL( m_dnSocket, 'Target_Room_Temp', GLOBAL_Target_Room_Temp );


	END_CASE

	state := state + 1;

	SysSockClose ( m_dnSocket );
	m_dnSocket := SOCKET_INVALID;


	m_error := 0;
END_FUNCTION_BLOCK

(* POU PLC_PRG, ST *)
PROGRAM PLC_PRG
VAR

	Need_init: BOOL := TRUE;


	Zinit:		Z033_INIT;
	Reader:	GET_DATA;

	z033Write:	Z033_WRITER;

	Read1W: DZ1W_READER;

	z033_temperature_set_old	: WORD;
	Uplink_Target_Temp_old		: WORD;

	z033_humidity_set_old		: WORD;
	Uplink_Target_Humid_old	: WORD;



END_VAR

(*
VAR RETAIN PERSISTENT
	GLOBAL_Target_Room_Temp: REAL;
END_VAR
*)
IF Need_init THEN


	z033_cmd := 255;
	z033_special_cmd := 255;

	mva8_0_cmd := 255;
	mva8_1_cmd := 255;
	mva8_2_cmd := 255;

	dz1w_cmd := 255;

	Zinit();
	z033Write();

	z033_temperature115_out := REAL_TO_WORD( GLOBAL_Target_Room_Temp );
	z033_hum116_out := REAL_TO_WORD( GLOBAL_Target_Room_Humid );


	Need_init := FALSE;
END_IF

(* TODO check if z033 really needs even parity. reprogram? *)


	Reader();
	Read1W();

	(* temp set *)

	IF (Reader.z033_temperature_set > SANE_TEMP_MIN) AND (Reader.z033_temperature_set < SANE_TEMP_MAX) AND (z033_temperature_set_old <> Reader.z033_temperature_set) THEN
		GLOBAL_Target_Room_Temp := Reader.z033_temperature_set;
		z033_temperature_set_old := Reader.z033_temperature_set;

		z033_temperature115_out := Reader.z033_temperature_set;

		Uplink_Target_Temp := REAL_TO_BYTE( GLOBAL_Target_Room_Temp );
		Uplink_Target_Temp_old := Uplink_Target_Temp;
	END_IF

	IF Uplink_Target_Temp_old <> Uplink_Target_Temp THEN
		GLOBAL_Target_Room_Temp := Uplink_Target_Temp;
		Uplink_Target_Temp_old := Uplink_Target_Temp;
	END_IF

	(* Fix crazy valiues *)

	IF GLOBAL_Target_Room_Temp < SANE_TEMP_MIN THEN
		GLOBAL_Target_Room_Temp := SANE_TEMP_MIN;
	END_IF

	IF GLOBAL_Target_Room_Temp > SANE_TEMP_MAX THEN
		GLOBAL_Target_Room_Temp := SANE_TEMP_MAX;
	END_IF


	(* humidity set *)



	IF (Reader.z033_humidity_set > SANE_HUMID_MIN) AND (Reader.z033_humidity_set < SANE_HUMID_MAX) AND (z033_humidity_set_old <> Reader.z033_humidity_set) THEN
		GLOBAL_Target_Room_Humid := Reader.z033_humidity_set;
		z033_humidity_set_old := Reader.z033_humidity_set;

		z033_hum116_out:= Reader.z033_humidity_set;

		Uplink_Target_Humid := REAL_TO_BYTE( GLOBAL_Target_Room_Humid );
		Uplink_Target_Humid_old := Uplink_Target_Humid;
	END_IF

	IF Uplink_Target_Humid_old <> Uplink_Target_Humid THEN
		GLOBAL_Target_Room_Humid := Uplink_Target_Humid;
		Uplink_Target_Humid_old := Uplink_Target_Humid;
	END_IF

	(* Fix crazy valiues *)

	IF GLOBAL_Target_Room_Humid < SANE_HUMID_MIN THEN
		GLOBAL_Target_Room_Humid := SANE_HUMID_MIN;
	END_IF

	IF GLOBAL_Target_Room_Humid > SANE_HUMID_MAX THEN
		GLOBAL_Target_Room_Humid := SANE_HUMID_MAX;
	END_IF


	(* TODO no net vars now, do it some other way *)
	(* Lower HUMIDITY in bathroom, if too high * )

	IF GLOBAL_Current_Bath_Air_Humid > GLOBAL_Target_Room_Humid THEN

		(* +10% of humidity = 100% of ventilation power *)
		Net_Ventilation_Request_Percent := REAL_TO_INT( MIN( 99, (GLOBAL_Current_Bath_Air_Humid - GLOBAL_Target_Room_Humid) * 10 ) );

	ELSE
		Net_Ventilation_Request_Percent := 0;
	END_IF
	*)





	z033Write();
END_PROGRAM

(* POU IO/Z033_INIT, ST *)
FUNCTION_BLOCK Z033_INIT
VAR_INPUT
END_VAR
VAR_OUTPUT
END_VAR
VAR
(*	SysRtcGetTime: DATE_AND_TIME; *)


END_VAR
	(* Set mode - const *)

	(*z033_Setup112 := 16#445B; *)
	z033_Setup112 :=
		2#111 OR (* vent speeds *)
		2#1000 OR (* Fan speed msg *)
		2#10000 OR (* Auto msg *)
		(* 2#1111100000 OR (* Possible modes *) *)
		2#0001100000 OR (* Heat or vent modes *)
		2#1110000000000 OR (* temp measure points *)
		(* 2#1110000000000000 (* hum measure points *) *)
		   2#0100000000000000 (* hum measure points - just ROOM *)
		;

	z033_Setup113 := 16#0714;

	z033_mode114_out := 2#01010001;

	z033_errmode11c_out := 0;

(*
	now := SysRtcGetTime();
*)
END_FUNCTION_BLOCK

(* POU IO/GET_DATA, ST *)
FUNCTION_BLOCK GET_DATA

VAR_INPUT
END_VAR

VAR_OUTPUT
	z033_temperature_set: WORD;
	z033_humidity_set: WORD;
	z033_room_temp: WORD;
	z033_mode: WORD;
	z033_vent_speed: WORD;
	z033_vent_auto: BOOL;
	z033_mode_vent: BOOL;
	z033_mode_heat: BOOL;
	z033_mode_cool: BOOL;
	z033_mode_humid: BOOL;
	z033_mode_dry: BOOL;
	mva_temperature: ARRAY[0..7] OF REAL;
END_VAR

VAR
     TEMP_REAL : REAL;
END_VAR
(* Gather all the data we need as input *)


(* Read from Z033 - check 'changed' bit first *)

IF (z033_errmode11c_in AND 16#1000) <> 0 THEN

	z033_errmode11c_out := 0; (* reset 'changed' bit and error state - TODO if we will use error state - handle it here too *)

	(* TODO read if we are initing *)


END_IF

	(* TODO read if changed, see above *)


	z033_mode := z033_mode114_in;
	z033_temperature_set := z033_temperature115_in; (* z033_temperature115_out := z033_temperature115_in; *)
	z033_humidity_set := z033_hum116_in;
	z033_room_temp	:= z033_room_temp117_in;

	z033_vent_speed := SHR( z033_mode, 1 ) AND 2#111;
	z033_vent_auto := (SHR( z033_mode, 3 ) AND 2#1) <> 0;

	z033_mode_vent := (SHR( z033_mode, 4 ) AND 2#1) <> 0;
	z033_mode_heat := (SHR( z033_mode, 5 ) AND 2#1) <> 0;
	z033_mode_cool := (SHR( z033_mode, 6 ) AND 2#1) <> 0;
	z033_mode_humid := (SHR( z033_mode, 7 ) AND 2#1) <> 0;
	z033_mode_dry := (SHR( z033_mode, 8 ) AND 2#1) <> 0;

	(* GLOBAL_Current_Dinner_Air_Temp := MIN_SANE_TEMP( z033_room_temp / 10.0, MVA0_t5 ) ; *)
	(* 0t5 = kitchen ceiling sensor, 1t5 = near floor down the window dinner room sensor *)

	(* GLOBAL_Current_Dinner_Air_Temp := MIN_SANE_TEMP( z033_room_temp / 10.0, MIN_SANE_TEMP( MVA0_t5, mva1_t3 ) ) ; *)
	GLOBAL_Current_Dinner_Air_Temp := AVG_SANE_TEMP3( z033_room_temp / 10.0, MVA0_t5, mva1_t3 );

	GLOBAL_Current_Dinner_Air_Bottom_Temp	:=	mva1_t3;
	GLOBAL_Current_Dinner_Air_Middle_Temp	:=	z033_room_temp / 10.0;
	GLOBAL_Current_Kitchen_Air_Ceiling_Temp	:=	MVA0_t5;
	GLOBAL_Current_Guest_Air_Temp := AVG_SANE_TEMP( mva2_t0, mva2_t1 ) ; (* guest room floor and ceiling (fire sensor) *)

	(* GLOBAL_Target_Room_Temp := z033_temperature_set; *)

	mva_temperature[0] := mva0_t0; (* 1/2 children floor *)
	mva_temperature[1] := mva0_t1; (* 1/2 children floor *)
	mva_temperature[2] := mva0_t2;	(* dinner floor *)
	mva_temperature[3] := mva0_t3;	(* entrance floor *)
	mva_temperature[4] := mva0_t4;	(* bath floor *)
	mva_temperature[5] := mva0_t5; (* Kitchen ceiling *)
	mva_temperature[6] := mva0_t6;
	mva_temperature[7] := mva0_t7; (* server room (equipment closet) top *)



	GLOBAL_Current_Children_Floor_Temp	:= MAX( mva0_t0, mva0_t1 );
	GLOBAL_Current_Dinner_Floor_Temp		:= mva0_t2;
	GLOBAL_Current_Entrance_Floor_Temp	:= mva0_t3;
	GLOBAL_Current_Bath_Floor_Temp		:= mva0_t4;

	GLOBAL_Current_Entrance_Air_Temp		:= MIN_SANE_TEMP( mva0_t7, mva0_t6 ); (* mva0_t7; (* currently in equipment closet *) *)

	GLOBAL_Current_Children_Air_Temp		:= MIN_SANE_TEMP( mva1_t0, mva1_t1 );

	GLOBAL_Current_Badroom_Air_Temp		:= mva1_t2;

	GLOBAL_Current_Bath_Air_Temp			:= 	mva1_t6;
	GLOBAL_Current_Bath_Tube_Temp		:= 	mva1_t7;

	TEMP_REAL	:= HUMID_CONV( V_In := mva1_t4 * 4 / 100, Zero_Off := 0.842, Slope := 0.031 );

	(* Sometimes we get insane value *)
	(* Assign sane data only *)
	IF (TEMP_REAL > 5) AND (TEMP_REAL < 95) THEN
		GLOBAL_Current_Bath_Air_Humid			:= LIMIT_VALUE( TEMP_REAL, 0, 100 );
	END_IF

	GLOBAL_Current_Outdoor_Air_Temp		:= mva1_t5;
END_FUNCTION_BLOCK

(* POU Conv/AVG_SANE_TEMP3, ST *)
FUNCTION AVG_SANE_TEMP3 : REAL

VAR_INPUT
	Ta, Tb, Tc : REAL;
END_VAR

VAR
	Ta_SANE, Tb_SANE, Tc_SANE : BOOL;
	Sum	: REAL;
	Count	: INT;
END_VAR
Ta_SANE := IS_SANE_TEMP( Ta );
Tb_SANE := IS_SANE_TEMP( Tb );
Tc_SANE := IS_SANE_TEMP( Tb );

Sum := 0;
Count :=0;

IF Ta_SANE THEN
	Sum := Sum + Ta;
	Count := Count + 1;
END_IF;

IF Tb_SANE THEN
	Sum := Sum + Tb;
	Count := Count + 1;
END_IF;

IF Tc_SANE THEN
	Sum := Sum + Tc;
	Count := Count + 1;
END_IF;

IF Count <= 0 THEN
	AVG_SANE_TEMP3 := -100; (* Surely insane low value *)
	RETURN;
END_IF

AVG_SANE_TEMP3 := Sum / Count;
END_FUNCTION

(* POU Conv/AVG_SANE_TEMP, ST *)
FUNCTION AVG_SANE_TEMP : REAL

VAR_INPUT
	Ta, Tb : REAL;
END_VAR

VAR
	Ta_SANE, Tb_SANE : BOOL;
END_VAR
Ta_SANE := IS_SANE_TEMP( Ta );
Tb_SANE := IS_SANE_TEMP( Tb );

IF Ta_SANE AND NOT Tb_SANE THEN
	AVG_SANE_TEMP := Ta;
	RETURN;
END_IF;

IF Tb_SANE AND NOT Ta_SANE THEN
	AVG_SANE_TEMP := Tb;
	RETURN;
END_IF;

IF Ta_SANE AND Tb_SANE THEN
	AVG_SANE_TEMP :=  (Ta + Tb) / 2;
	RETURN;
END_IF;


	AVG_SANE_TEMP := SANE_TEMP_MIN-100; (* Surely insane low value *)
END_FUNCTION

(* POU Conv/MIN_SANE_TEMP, ST *)
FUNCTION MIN_SANE_TEMP : REAL

VAR_INPUT
	Ta, Tb : REAL;
END_VAR

VAR
	Ta_SANE, Tb_SANE : BOOL;
END_VAR
Ta_SANE := IS_SANE_TEMP( Ta );
Tb_SANE := IS_SANE_TEMP( Tb );

IF Ta_SANE AND NOT Tb_SANE THEN
	MIN_SANE_TEMP := Ta;
	RETURN;
END_IF;

IF Tb_SANE AND NOT Ta_SANE THEN
	MIN_SANE_TEMP := Tb;
	RETURN;
END_IF;

IF Ta_SANE AND Tb_SANE THEN
	MIN_SANE_TEMP := MIN( Ta, Tb );
	RETURN;
END_IF;


	MIN_SANE_TEMP := SANE_TEMP_MIN-100; (* Surely insane low value *)
END_FUNCTION

(* POU Conv/HUMID_CONV, ST *)
FUNCTION HUMID_CONV : REAL

VAR_INPUT
	V_In		:	REAL;

	Zero_Off	:	REAL;
	Slope		:	REAL;
END_VAR

VAR
END_VAR
	HUMID_CONV := (V_In - Zero_Off) / Slope;
END_FUNCTION

(* POU IO/Z033_WRITER, ST *)
FUNCTION_BLOCK Z033_WRITER

VAR_INPUT
	Enforce : BOOL := FALSE;

	z033_vent_speed: WORD;
	z033_vent_auto: BOOL := TRUE;
	z033_mode_vent: BOOL;
	z033_mode_heat: BOOL := TRUE;
	z033_mode_cool: BOOL;
	z033_mode_humid: BOOL;
	z033_mode_dry: BOOL;



	(* z033_floor_temp: REAL; *)
	z033_outdoor_hum: REAL;
	z033_room_hum: REAL;
	z033_air_hum: REAL;
END_VAR

VAR_OUTPUT
END_VAR

VAR
	z033_mode: WORD;
	z033_mode_old: WORD;
	TEMP: WORD;
	z033_outdoor_hum119_out_old: WORD;
	z033_room_hum11a_out_old: WORD;
	z033_air_hum11b_out_old: WORD;

	z033_floor_temp118_out_old: REAL;
	z033_air_temp_117_out_old: REAL;

	GLOBAL_Target_Room_Temp_old: WORD;

	GLOBAL_Target_Room_Humid_old : WORD;
	GLOBAL_Current_Bath_Air_Humid_old: WORD;

	(* Set actual date and time *)

	(* z033_DateTime, Minutes, Hours, WeekDay: WORD; *)

	z033_DateTime				: WORD;
	systime						: SysTime64;
	now							: SystemTimeDate;
	TimeReader					: CurTimeEx;

END_VAR
(* Write current values to Z033 panel *)

	z033_mode := 1; (* lower bit - panel is on *)

	z033_mode := z033_mode OR SHL(z033_vent_speed AND 2#111, 1);

	IF z033_vent_auto THEN
		z033_mode := z033_mode OR 2#10000;
	END_IF

	IF z033_mode_vent THEN
		z033_mode := z033_mode OR 2#100000;
	END_IF

	IF z033_mode_heat THEN
		z033_mode := z033_mode OR 2#1000000;
	END_IF

	IF z033_mode_cool THEN
		z033_mode := z033_mode OR 2#10000000;
	END_IF

	IF z033_mode_humid THEN
		z033_mode := z033_mode OR 2#100000000;
	END_IF

	IF z033_mode_dry THEN
		z033_mode := z033_mode OR 2#1000000000;
	END_IF


	IF z033_mode <> z033_mode_old THEN
		z033_mode114_out := z033_mode;
		z033_mode_old := z033_mode;
	END_IF

(*
	TEMP := REAL_TO_WORD( z033_outdoor_hum * 10 );

	IF TEMP <> z033_outdoor_hum119_out_old THEN
		z033_outdoor_hum119_out := TEMP;
		z033_outdoor_hum119_out_old := TEMP;
	END_IF


	TEMP := REAL_TO_WORD( z033_room_hum * 10 );

	IF TEMP <> z033_room_hum11a_out_old THEN
		z033_room_hum11a_out := TEMP;
		z033_room_hum11a_out_old := TEMP;
	END_IF



	TEMP := REAL_TO_WORD( z033_air_hum * 10 );

	IF TEMP <> z033_air_hum11b_out_old THEN
		z033_air_hum11b_out := TEMP;
		z033_air_hum11b_out_old := TEMP;
	END_IF
*)

	IF z033_floor_temp118_out_old <> GLOBAL_Current_Dinner_Floor_Temp THEN
		z033_floor_temp118_out := REAL_TO_WORD( GLOBAL_Current_Dinner_Floor_Temp * 10 );
		z033_floor_temp118_out_old := GLOBAL_Current_Dinner_Floor_Temp;
	END_IF

	(* temp off - wrong
	IF z033_temperature115_out_old <> GLOBAL_Current_Dinner_Air_Temp THEN
		z033_temperature115_out := REAL_TO_WORD( GLOBAL_Current_Dinner_Air_Temp * 10 );
		z033_temperature115_out_old := GLOBAL_Current_Dinner_Air_Temp;
	END_IF
	*)

	(* temp replacement *)
	IF z033_air_temp_117_out_old <> GLOBAL_Current_Entrance_Air_Temp THEN
		z033_air_temp_117_out := REAL_TO_WORD( GLOBAL_Current_Entrance_Air_Temp * 10 );
		z033_air_temp_117_out_old := GLOBAL_Current_Entrance_Air_Temp;
	END_IF





	TEMP := REAL_TO_WORD( GLOBAL_Target_Room_Temp  );

	IF TEMP <> GLOBAL_Target_Room_Temp_old THEN
		z033_temperature115_out := TEMP;
		GLOBAL_Target_Room_Temp_old := TEMP;
	END_IF


	(* Humidity *)

	TEMP := REAL_TO_WORD( GLOBAL_Target_Room_Humid  );

	(* hum target *)
	IF TEMP <> GLOBAL_Target_Room_Humid_old THEN
		z033_hum116_out := TEMP;
		GLOBAL_Target_Room_Humid_old := TEMP;
	END_IF



	TEMP := REAL_TO_WORD( GLOBAL_Current_Bath_Air_Humid  );

	IF TEMP <> GLOBAL_Current_Bath_Air_Humid_old THEN
		z033_room_hum11a_out := TEMP * 10;
		GLOBAL_Current_Bath_Air_Humid_old := TEMP;
	END_IF


	(* Set actual date and time *)

	now.Day :=0;
	now.DayOfWeek :=0;
	now.dwHighMsec :=0;
	now.dwLowMSecs :=0;
	now.Milliseconds :=0;
	now.Minute :=0;
	now.Second :=0;
	now.Hour :=0;
	now.Year :=0;
	now.Month :=0;

	systime.ulHigh :=0;
	systime.ulLow :=0;

	TimeReader( SystemTime := systime, TimeDate:= now );


	z033_DateTime := 0;

	z033_DateTime := 	UINT_TO_WORD(now.Hour) AND 2#011111;


(*
	z033_DateTime := 	z033_DateTime OR ( SHL( UINT_TO_WORD(now.Minute) ,5) AND 2#011111100000 );
	z033_DateTime := 	z033_DateTime OR ( SHL( UINT_TO_WORD(now.DayOfWeek-1),11) AND 2#011100000000000 );
*)
	z033_DateTime := 	z033_DateTime OR ( SHL( 2#0111111 AND UINT_TO_WORD(now.Minute) ,5)  );
	z033_DateTime := 	z033_DateTime OR ( SHL( 2#0000111 AND UINT_TO_WORD(now.DayOfWeek-1),11)  );



	z033_clock11d_out := z033_DateTime;
END_FUNCTION_BLOCK

(* POU IO/DZ1W_READER, ST *)
FUNCTION_BLOCK DZ1W_READER

VAR_INPUT
END_VAR

VAR_OUTPUT

	sensor_temp : ARRAY [0..15] OF REAL;

END_VAR

VAR
END_VAR
sensor_temp[0] := Word4Fract( sensor_id0 );
sensor_temp[1] := Word4Fract( sensor_id1);
sensor_temp[2] := Word4Fract( sensor_id2);
sensor_temp[3] := Word4Fract( sensor_id3);
sensor_temp[4] := Word4Fract( sensor_id4);
sensor_temp[5] := Word4Fract( sensor_id5);
sensor_temp[6] := Word4Fract( sensor_id6);
sensor_temp[7] := Word4Fract( sensor_id7);

(*
sensor_temp[8] := Word4Fract( sensor_id8);
sensor_temp[9] := Word4Fract( sensor_id9);
sensor_temp[10] := Word4Fract( sensor_id10);
sensor_temp[11] := Word4Fract( sensor_id11);
sensor_temp[12] := Word4Fract( sensor_id12);
sensor_temp[13] := Word4Fract( sensor_id13);
sensor_temp[13] := Word4Fract( sensor_id14);
sensor_temp[15] := Word4Fract( sensor_id15);
*)
END_FUNCTION_BLOCK

(* POU Conv/Word4Fract, ST *)
FUNCTION Word4Fract : REAL
VAR_INPUT
	IN : WORD;
END_VAR
VAR
END_VAR
Word4Fract := WORD_TO_REAL(IN) / 16.0;
END_FUNCTION

(* POU MQTT_UDP/MQTT_MAIN, ST *)
PROGRAM MQTT_MAIN

VAR

	SocketHandle: 	DINT	:= SOCKET_INVALID; (* descriptor of open Socket *)
	addr:				SOCKADDRESS;
	flags:				DINT := 0;
	(*buf:				STRING;
	pkt_size:			DINT := 0;*)

	pkt :				MAKE_MQTT_PKT;

END_VAR
RETURN; (* turn off *)

IF SocketHandle <> SOCKET_INVALID THEN
	SocketHandle := SysSockCreate( SOCKET_AF_INET, SOCKET_DGRAM, SOCKET_IPPROTO_UDP );
END_IF

IF SocketHandle <> SOCKET_INVALID THEN
	RETURN;
END_IF

addr.sin_family := SOCKET_AF_INET;
addr.sin_port :=1883; (* MQTT UDP *)
addr.sin_addr := SOCKET_INADDR_BROADCAST;

pkt( topic := 'plc_topic', data := 'plc_val' );

SysSockSendTo( SocketHandle, ADR(pkt.buf), pkt.LEN, flags, ADR(addr),   SIZEOF(addr)  );
END_PROGRAM

(* POU MQTT_UDP/MAKE_MQTT_PKT, ST *)
FUNCTION_BLOCK MAKE_MQTT_PKT
VAR_INPUT
	topic : STRING;
	data : STRING;
END_VAR

VAR_OUTPUT
	buf :	STRING;
	len : 	DINT;
END_VAR

VAR
(*	blen :	DINT; *)
	tlen :	DINT;
	dlen :	DINT;
	total : 	DINT;
END_VAR
	tlen := LEN(topic);
	dlen :=LEN(data);

	INSERT( buf, '$30', 0 ); (* 'publish' pkt type *)

	total := tlen + dlen + 2; (* packet size *)

	tlen := SHR( tlen, 8 ) ;

	buf := CONCAT( buf, CHR_TO_STRING( DINT_TO_BYTE( SHR( tlen, 8 ) ) )  );
	buf := CONCAT( buf, CHR_TO_STRING( DINT_TO_BYTE( tlen ) ) );

	buf := CONCAT( buf, topic );
	buf := CONCAT( buf, data );

	(* MAKE_MQTT_PKT := buf; *)

	LEN := total + 2; (* ERROR - supposed that pkt len < 128 and len is one byte *)
END_FUNCTION_BLOCK

(* POU Conv/DALLAS_CONV, ST *)
FUNCTION DALLAS_CONV : REAL

VAR_INPUT
	T	: WORD;
END_VAR

VAR
END_VAR
DALLAS_CONV := WORD_TO_REAL(T) / 16.0;
END_FUNCTION

(* POU MQTT_UDP/PACK_LEN, ST *)
FUNCTION PACK_LEN : STRING
VAR_INPUT
	data_len : DINT;
END_VAR
VAR
	out : STRING := '';
	b : BYTE;
END_VAR
WHILE TRUE DO


        B := DINT_TO_BYTE( data_len MOD 128 );
        data_len := data_len / 128;

        IF data_len > 0 THEN
            B := B OR DINT_TO_BYTE( 16#80 );
	END_IF

        out := CONCAT( out, CHR_TO_STRING(b) );

        IF( data_len = 0 ) THEN
		EXIT;
	END_IF
END_WHILE

PACK_LEN := out;
END_FUNCTION
